Omron CX-Programmer project NuevoProyecto (CX-Programmer ?)

# PLC trabajoGrafcet: CPM1(CPM1A) CPU30

## Program NuevoPrograma1 (no task)
Local symbols
CNT_A BOOL
TIM_A BOOL
TIM_B BOOL

### Section Sección1

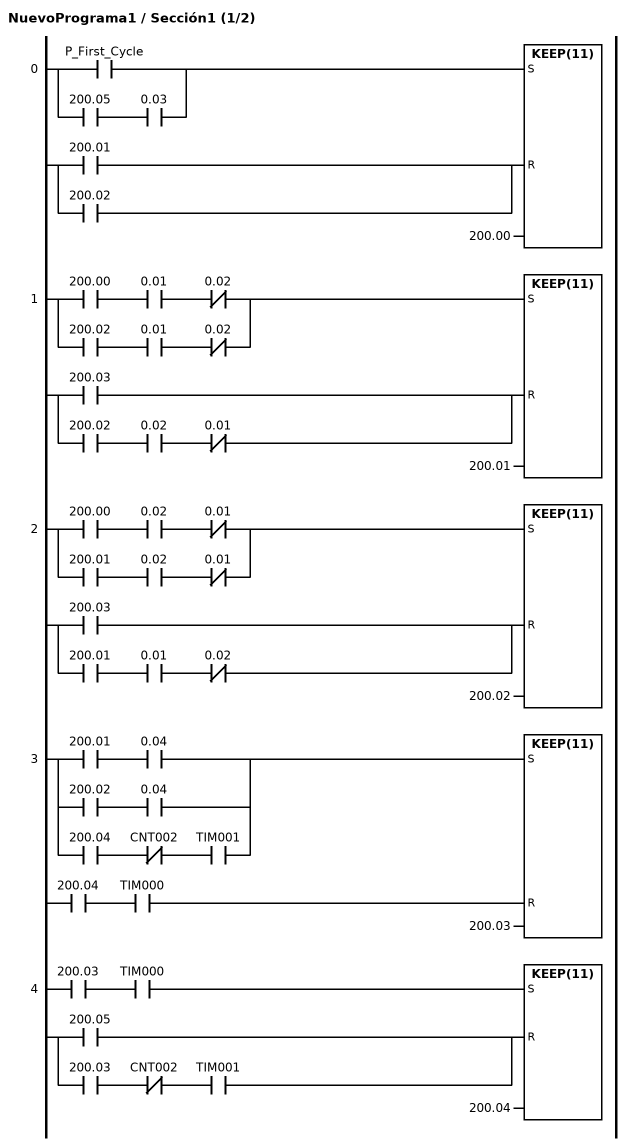
; rung 0
LD P_First_Cycle
LD 200.05
AND 0.03
ORLD
LD 200.01
OR 200.02
KEEP(11) 200.00
; rung 1
LD 200.00
AND 0.01
ANDNOT 0.02
LD 200.02
AND 0.01
ANDNOT 0.02
ORLD
LD 200.03
LD 200.02
AND 0.02
ANDNOT 0.01
ORLD
KEEP(11) 200.01
; rung 2
LD 200.00
AND 0.02
ANDNOT 0.01
LD 200.01
AND 0.02
ANDNOT 0.01
ORLD
LD 200.03
LD 200.01
AND 0.01
ANDNOT 0.02
ORLD
KEEP(11) 200.02
; rung 3
LD 200.01
AND 0.04
LD 200.02
AND 0.04
ORLD
LD 200.04
ANDNOT CNT002
AND TIM001
ORLD
LD 200.04
AND TIM000
KEEP(11) 200.03
; rung 4
LD 200.03
AND TIM000
LD 200.05
LD 200.03
ANDNOT CNT002
AND TIM001
ORLD
KEEP(11) 200.04

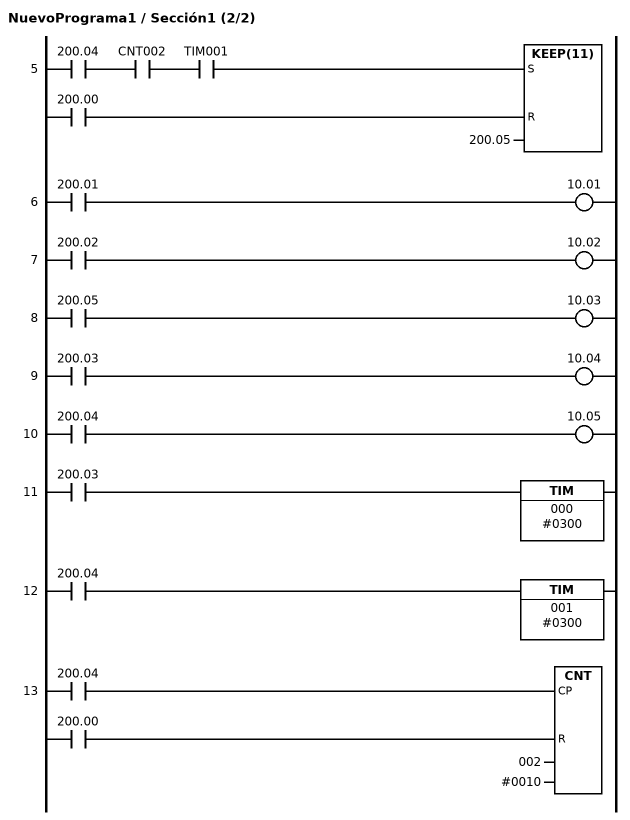
; rung 5
LD 200.04
AND CNT002
AND TIM001
LD 200.00
KEEP(11) 200.05
; rung 6
LD 200.01
OUT 10.01
; rung 7
LD 200.02
OUT 10.02
; rung 8
LD 200.05
OUT 10.03
; rung 9
LD 200.03
OUT 10.04
; rung 10
LD 200.04
OUT 10.05
; rung 11
LD 200.03
TIM 000 #0300
; rung 12
LD 200.04
TIM 001 #0300
; rung 13
LD 200.04
LD 200.00
CNT 002 #0010
; rung 14
END(01)